{attribute 'GeneratedUsingTerminal: EK1100-0000-0018'}
{attribute addProperty BoxType "EK1100-0000-0018"}
{attribute addProperty Id "Beckhoff_CUxxxxEK1122Beckhoff_CUxxxxEK1122_FDB340FF126"}
{attribute addProperty CRC "448715056"}
{attribute addProperty Size "126"}
TYPE Beckhoff_CUxxxx_1ABED930 EXTENDS EK1100_AB5A9467 :
STRUCT
	{attribute addProperty Name "Beckhoff_CUxxxxEK1122"}
	{attribute addProperty PreviousPort "Beckhoff CUxxxx : B"}
	Beckhoff_CUxxxxEK1122 : Beckhoff_CUxxxxEK1122_FDB340FF;
END_STRUCT
END_TYPE

(* stored: Version 1.2.0.0, ProductVersion 3.1.4024.9
   DUT Beckhoff_CUxxxx_1ABED930: Id {c78af9da-cc5d-49bc-b297-97fd49302663} *)
